// Mitsubishi GX Works2 project: jumpEx01   PLC: Q02/Q02H

PROGRAM MAIN
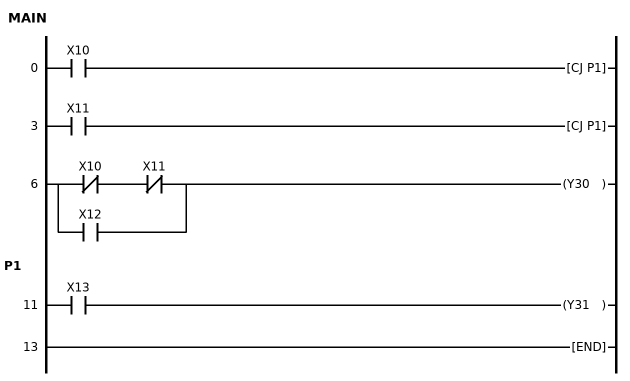
0     LD      X10
      CJ      P1
3     LD      X11
      SCJ     P1
6     LDI     X10
      ANI     X11
      OR      X12
      OUT     Y30
      P1
11    LD      X13
      OUT     Y31
13    END
END_PROGRAM
